(* IEC 61131-3 sources: inproshop/Team-Test6_exported/1.Function/FB/Mode(模式), 6 files *)

(* ---- Str_Machine.st ---- *)
TYPE Str_Machine :
STRUCT
	OP_Emg_Stop		:BOOL;//操作面板紧急停止按钮
	OP_StartButton	:BOOL;//操作面板启动按钮
	OP_StopButton	:BOOL;//操作面板停止按钮
	OP_ResetButton	:BOOL;//操作面板复位按钮
	OP_AutoManual	:BOOL;//操作面板手/自动选择
	EmgSafetyRelay	:BOOL;//急停安全继电器信号
	SafetyDoorRelay	:BOOL;//安全门安全继电器信号
	LightCurtainRelay:BOOL;//光栅安全继电器信号
	AirPresure		:BOOL;//气源压力开关信号
	RedLightHouse	:BOOL;//红色灯塔
	YeLightHouse	:BOOL;//黄色灯塔
	GrLightHouse	:BOOL;//绿色灯塔
	Buzzer			:BOOL;//蜂鸣器
	StartLamp		:BOOL;//开始按钮灯
	StopLamp		:BOOL;//停止按钮灯
	ResetLamp		:BOOL;//复位按钮灯
	Light			:BOOL;//日光灯
	Emg_Stop		:ARRAY[0..9]OF BOOL := [10(TRUE)];//急停信号
	LightCurtain	:ARRAY[0..9]OF BOOL := [10(TRUE)];//安全光栅信号
	SafetyDoor		:ARRAY[0..9]OF BOOL := [10(TRUE)];//安全门信号
	Speed			:REAL;//设备运行速率
	CycleTime		:Str_CycleTime;//周期时间
	PowerOnTime		:UDINT;//开机时间
	RunTime			:UDINT;//运行时间
	EfficencyResult	:REAL;//设备稼动率
	EfficencyClear	:BOOL;//稼动率清零
END_STRUCT
END_TYPE

(* ---- Str_Mode.st ---- *)
TYPE Str_Mode :
STRUCT
	Cmd:Str_ModeCmd;//控制
	Status:Str_ModeStatus;//状态
	Out:Str_ModeOut;//输出控制
END_STRUCT
END_TYPE

(* ---- Str_ModeCmd.st ---- *)
TYPE Str_ModeCmd :
STRUCT
	AutoManualButton:BOOL;//手自动按钮
	RunButton		:BOOL;//启动按钮
	StopButton		:BOOL;//停止按钮
	ResetButton		:BOOL;//复位按钮
	CycleEndButton	:BOOL;//周期停止按钮
	StepButton		:BOOL;//单步按钮
	HomingButton	:BOOL;//回原按钮
	NullPartButton	:BOOL;//空跑按钮
	OfflineButton	:BOOL;//离线按钮
	LampTest		:BOOL;//灯光测试
	Debug_BUZButton	:BOOL;//蜂鸣器屏蔽
	SafetyDoorShieild:BOOL;//安全门屏蔽
	NullPartRunLine	:BOOL;//空托盘跑线
	ManUnlock		:BOOL;//互锁信号解锁
END_STRUCT
END_TYPE

(* ---- Str_ModeOut.st ---- *)
TYPE Str_ModeOut :
STRUCT

	HomeStart:BOOL;//设备初始化开始
	ErrorReset:BOOL;//设备报警复位
	Stop:BOOL;//设备停止
	AutoRun_R:BOOL;//运转中上升沿
	AutoRun_F:BOOL;// 运转中下降沿
	HomeOK_R:BOOL;//回原完成上升沿
	HomeOK_F:BOOL;//回原完成下降沿
	HomeStart_R:BOOL;//回原开始上升沿
	HomeStart_F:BOOL;//回原开始下降沿
END_STRUCT
END_TYPE

(* ---- Str_ModeStatus.st ---- *)
TYPE Str_ModeStatus :
STRUCT
	ManualMode	:BOOL;//手动模式
	AutoMode	:BOOL;//自动模式
	RunMode		:BOOL;//运转模式
	StopMode	:BOOL;//停止模式
	CycleMode	:BOOL;//周期模式
	StepMode	:BOOL;//单步模式
	DryMode		:BOOL;//空跑模式
	ClearMode	:BOOL;//清料模式
	OfflineMode	:BOOL;//离线模式
	HandMode	:BOOL;//人工模式
	StationMode	:BOOL;//单工位运行模式
	AutoRunning	:BOOL;//自动运转中
	StepRunning	:BOOL;//单步运转中
	HomeOK		:BOOL;//初始化完成
	EStop		:BOOL;//急停
	Fault		:BOOL;//报警
	Warning		:BOOL;//警告

END_STRUCT
END_TYPE

(* ---- FB_ModeControl_V1.st ---- *)
FUNCTION_BLOCK FB_ModeControl_V1
VAR_INPUT
	iClock:Str_Clock;//系统时钟
	iStartDelay:TIME;//延时启动
	iEstop:BOOL;//急停报警
	iAlam:BOOL;//暂停报警
	iWarn:BOOL;//警告
END_VAR
VAR_IN_OUT
	ioMachine:Str_Machine;//设备
	ioMode:Str_Mode;//模式
END_VAR
VAR_OUTPUT
END_VAR
VAR
	i:INT;//循环变量
	Start_R:R_TRIG;//开始按钮上升沿
	Reset_R:R_TRIG;//复位按钮上升沿
	Step_R:R_TRIG;//单步按钮上升沿
	Home_R:R_TRIG;//回原按钮上升沿
	Home_F:F_TRIG;//回原按钮下降沿
	DelayStart:TON;//开始按钮延时
	DelayReset:TON;//复位按钮延时
	DelayStop:TON;//停止按钮延时
	AutoRun_R:R_TRIG;//运转中上升沿
	AutoRun_F:F_TRIG;//运转中上升沿
	HomeOK_R:R_TRIG;//回原完成上升沿
	HomeOK_F:F_TRIG;//回原完成下降沿
	HomeStart_R:R_TRIG;//回原开始上升沿
	HomeStart_F:F_TRIG;//回原开始下降沿
END_VAR

//******************************************************HMI&Machine&Interface控制状态切换

//启动按钮状态获取
Start_R(CLK:=DelayStart.Q );//上升沿
DelayStart(IN:=ioMachine.OP_StartButton OR ioMode.Cmd.RunButton,PT:=iStartDelay);//延时启动
//复位按钮状态获取
Reset_R(CLK:=ioMachine.OP_ResetButton OR ioMode.Cmd.ResetButton OR ioMode.Cmd.HomingButton);//上升沿
DelayReset(IN:=ioMachine.OP_ResetButton OR ioMode.Cmd.ResetButton,PT:=T#3S);//复位按钮延时
//停止按钮状态获取
DelayStop(IN:=ioMachine.OP_StopButton OR ioMode.Cmd.StopButton,PT:=T#3S);//停止延时
//单步按钮状态获取
Step_R(CLK:=ioMode.Cmd.StepButton);
//回原按钮状态获取
Home_R(CLK:=ioMode.Cmd.HomingButton OR DelayReset.Q);
Home_F(CLK:=ioMode.Cmd.HomingButton OR DelayReset.Q);

//报警&警告状态切换
ioMode.Status.EStop:=iEstop;
ioMode.Status.Fault:=iEstop OR iAlam;
ioMode.Status.Warning:=iWarn;

IF Reset_R.CLK THEN
	ioMode.Out.ErrorReset:=TRUE;
ELSE
	ioMode.Out.ErrorReset:=FALSE;
END_IF;

IF DelayStop.IN OR ioMode.Status.Fault OR ioMode.Status.EStop THEN
	ioMode.Out.Stop:=TRUE;
ELSE
	ioMode.Out.Stop:=FALSE;
END_IF;

//手自动模式切换
ioMode.Status.ManualMode:=NOT ioMachine.OP_AutoManual;
ioMode.Status.AutoMode:=ioMachine.OP_AutoManual;

//手动互锁条件屏蔽复位
IF ioMode.Status.AutoMode THEN
	ioMode.Cmd.ManUnlock:=FALSE;
END_IF;

//回原
IF Home_R.Q THEN
	ioMode.Status.HomeOK:=FALSE;
END_IF
IF ioMode.Status.AutoMode AND NOT ioMode.Status.Fault AND Home_F.Q AND NOT ioMode.Status.AutoRunning THEN
	ioMode.Out.HomeStart:=TRUE;
END_IF;

IF ioMode.Status.Fault OR DelayStop.IN OR ioMode.Status.ManualMode OR ioMode.Status.HomeOK THEN
	ioMode.Out.HomeStart:=FALSE;
END_IF;

IF iEstop OR DelayStop.Q THEN
	ioMode.Status.HomeOK:=FALSE;
END_IF;

//运转中
IF ioMode.Status.HomeOK AND ioMode.Status.AutoMode AND Start_R.Q THEN
	ioMode.Status.AutoRunning:=TRUE;
END_IF;
IF ioMode.Status.Fault OR DelayStop.IN OR ioMode.Status.ManualMode OR Home_R.Q THEN
	ioMode.Status.AutoRunning:=FALSE;
END_IF;

//单步模式
IF ioMode.Status.StepMode THEN
	ioMode.Status.StepRunning:=FALSE;
END_IF;
IF Start_R.Q THEN
	ioMode.Status.StepRunning:=TRUE;
END_IF;

//状态沿获取
AutoRun_R(CLK:= ioMode.Status.AutoRunning, Q=>ioMode.Out.AutoRun_R );
AutoRun_F(CLK:= ioMode.Status.AutoRunning, Q=>ioMode.Out.AutoRun_F );
HomeOK_R(CLK:= ioMode.Status.HomeOK, Q=>ioMode.Out.HomeOK_R );
HomeOK_F(CLK:= ioMode.Status.HomeOK, Q=>ioMode.Out.HomeOK_F );
HomeStart_R(CLK:= ioMode.Out.HomeStart, Q=>ioMode.Out.HomeStart_R );
HomeStart_F(CLK:= ioMode.Out.HomeStart, Q=>ioMode.Out.HomeStart_F );

(*************************************************指示灯控制*********************************************************)
//上电&测试点亮塔灯按钮灯
IF iClock.FirstRun OR ioMode.Cmd.LampTest THEN
	ioMachine.RedLightHouse:=TRUE;
	ioMachine.YeLightHouse:=TRUE;
	ioMachine.GrLightHouse:=TRUE;
	ioMachine.StartLamp:=TRUE;
	ioMachine.StopLamp:=TRUE;
	ioMachine.ResetLamp:=TRUE;
	ioMachine.Light:=TRUE;
ELSE
	ioMachine.RedLightHouse:=FALSE;
	ioMachine.YeLightHouse:=FALSE;
	ioMachine.GrLightHouse:=FALSE;
	ioMachine.StartLamp:=FALSE;
	ioMachine.StopLamp:=FALSE;
	ioMachine.ResetLamp:=FALSE;
	ioMachine.Buzzer:=FALSE;
END_IF;

IF ioMode.Status.Fault THEN//停止类报警发生时，停止按钮灯亮，红色塔灯、蜂鸣器、复位按钮灯闪烁
	ioMachine.StopLamp:=TRUE;
	IF iClock.Clock_1s THEN
		ioMachine.RedLightHouse:=TRUE;
		ioMachine.Buzzer:=TRUE;
		ioMachine.ResetLamp:=TRUE;
	END_IF;
ELSIF iOMode.Status.Warning AND ioMode.Status.AutoRunning THEN//自动运转中，发生不停机报警时，绿色塔灯、开始按钮灯亮，黄色塔灯、蜂鸣器1S+0.2S闪烁,复位按钮灯1S闪烁
	ioMachine.StartLamp:=TRUE;
	ioMachine.GrLightHouse:=TRUE;
	IF iClock.Clock_1s AND iClock.Clock_100ms THEN
		ioMachine.YeLightHouse:=TRUE;
		ioMachine.Buzzer:=TRUE;
	END_IF;
	IF iClock.Clock_1s THEN
		ioMachine.ResetLamp:=TRUE;
	END_IF;
ELSIF ioMode.Status.AutoMode AND ioMode.Status.HomeOK AND NOT ioMode.Status.Fault AND NOT ioMode.Status.AutoRunning AND NOT DelayStart.IN THEN//自动模式下，原点回归完成，无报警时，绿色按钮灯闪烁
	ioMachine.StopLamp:=TRUE;
	ioMachine.YeLightHouse:=TRUE;
	IF iClock.Clock_1s THEN
		ioMachine.StartLamp:=TRUE;
	END_IF;
ELSIF ioMode.Status.AutoMode AND ioMode.Status.HomeOK AND NOT ioMode.Status.Fault AND NOT ioMode.Status.AutoRunning AND  DelayStart.IN THEN//自动模式下，原点回归完成，无报警时，绿色按钮灯闪烁
	ioMachine.StopLamp:=TRUE;
	ioMachine.YeLightHouse:=TRUE;
	IF iClock.Clock_1s THEN
		ioMachine.StartLamp:=TRUE;
	END_IF;
	IF  iClock.Clock_100ms THEN
		ioMachine.YeLightHouse:=TRUE;
		ioMachine.Buzzer:=TRUE;
	END_IF;
ELSIF ioMode.Status.AutoMode AND NOT ioMode.Status.HomeOK AND NOT ioMode.Status.Fault AND NOT iOMode.Status.AutoRunning AND NOT ioMode.Out.HomeStart  THEN//自动模式下，原点回归未完成，无报警时，黄色按钮灯亮
	ioMachine.StopLamp:=TRUE;
	ioMachine.YeLightHouse:=TRUE;
	ioMachine.ResetLamp:=TRUE;
ELSIF ioMode.Status.ManualMode AND  NOT ioMode.Status.Fault THEN//手动模式下，设备未初始化，设备未报警时，停止按钮灯、红色塔灯亮
	ioMachine.StopLamp:=TRUE;
	ioMachine.RedLightHouse:=TRUE;
ELSIF ioMode.Out.HomeStart THEN//初始化中开始按钮灯亮，绿色塔灯1S闪烁
	ioMachine.StartLamp:=TRUE;
	IF iClock.Clock_1s THEN
		ioMachine.GrLightHouse:=TRUE;
	END_IF;
ELSIF  iOMode.Status.AutoRunning THEN//自动运转中，开始按钮灯、绿色塔灯亮
	ioMachine.StartLamp:=TRUE;
	ioMachine.GrLightHouse:=TRUE;

ELSE//其他情况塔灯闪烁
	IF iClock.Clock_1s THEN
		ioMachine.RedLightHouse:=TRUE;
		ioMachine.YeLightHouse:=TRUE;
		ioMachine.GrLightHouse:=TRUE;
	END_IF;
END_IF;
//蜂鸣器屏蔽
IF ioMode.Cmd.Debug_BUZButton THEN
	ioMachine.Buzzer:=FALSE;
END_IF;
//复位后蜂鸣器屏蔽取消
// IF ioMode. Out.ErrorReset THEN
// 	ioMode.Cmd.Debug_BUZButton:=FALSE;
// END_IF

(*************************安全信号汇总**************************************)
//急停按钮
FOR i:=0 TO 9 BY 1 DO
	IF NOT ioMachine.Emg_Stop[i] THEN
		ioMachine.EmgSafetyRelay:=FALSE;
		EXIT;
	END_IF;
	ioMachine.EmgSafetyRelay:=TRUE;
END_FOR;

//安全门
FOR i:=0 TO 9 BY 1 DO
	IF NOT ioMachine.SafetyDoor[i] AND NOT ioMode.Cmd.SafetyDoorShieild THEN
		ioMachine.SafetyDoorRelay:=FALSE;
		EXIT;
	END_IF;
	ioMachine.SafetyDoorRelay:=TRUE;
END_FOR;

//安全光栅
FOR i:=0 TO 9 BY 1 DO
	IF NOT ioMachine.LightCurtain[i] THEN
		ioMachine.LightCurtainRelay:=FALSE;
		EXIT;
	END_IF;
	ioMachine.LightCurtainRelay:=TRUE;
END_FOR;

(*************************整机CT计时**************************************)
IF ioMode.Status.AutoRunning THEN
	IF ioMachine.CycleTime.Start THEN
		ioMachine.CycleTime.Start:= FALSE;
		ioMachine.CycleTime.Befor:=ioMachine.CycleTime.Now;
		ioMachine.CycleTime.Now:=0;
	END_IF;

	IF iClock.Clock_100ms_R THEN
		ioMachine.CycleTime.Now:=ioMachine.CycleTime.Now+1;
	END_IF;
END_IF;

(*************************整机稼动率统计**************************************)
//开机时间统计
//运行时间统计
IF iClock.Clock_1s_R THEN
	ioMachine.PowerOnTime:=ioMachine.PowerOnTime+1;
	IF ioMode.Status.AutoRunning THEN
		ioMachine.RunTime:=ioMachine.RunTime+1;
	END_IF;
END_IF;

IF ioMachine.PowerOnTime<>0 THEN
	ioMachine.EfficencyResult:=UDINT_TO_REAL(ioMachine.RunTime)/UDINT_TO_REAL(ioMachine.PowerOnTime);
ELSE
	ioMachine.EfficencyResult:=0;
END_IF;
IF ioMachine.EfficencyClear THEN
	ioMachine.PowerOnTime:=0;
	ioMachine.RunTime:=0;
	ioMachine.EfficencyClear:=FALSE;
END_IF;

//整机速度限制
IF ioMachine.Speed <= 0 OR ioMachine.Speed > 100 THEN
	ioMachine.Speed:=10;
END_IF
